FUNCTION_BLOCK CmdWaterDischargeSLBLogicBasic (* Basic Function Block Type *)
  (* Standard: 61499-2 *)
  (* Version 0.0, 7/31/2024, Administrator, Schneider Electric, Template *)
  PACKAGE SE.Nereda;
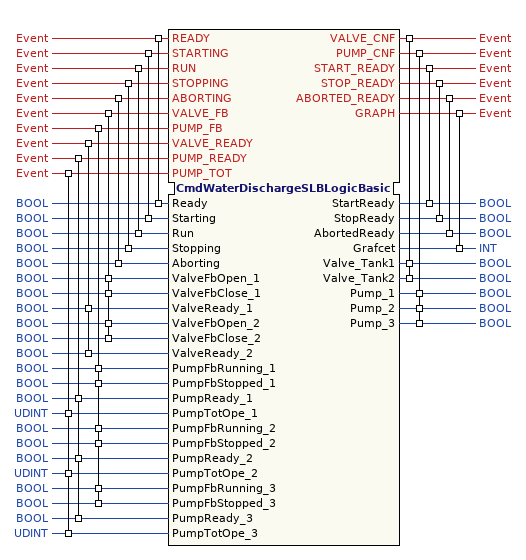
  EVENT_INPUT
    READY WITH Ready;
    STARTING WITH Starting; (* Normal Execution Request *)
    RUN WITH Run;
    STOPPING WITH Stopping;
    ABORTING WITH Aborting;
    VALVE_FB WITH ValveFbOpen_1, ValveFbClose_1, ValveFbOpen_2, ValveFbClose_2;
    PUMP_FB WITH PumpFbRunning_1, PumpFbStopped_1, PumpFbRunning_2, PumpFbStopped_2, PumpFbRunning_3, PumpFbStopped_3;
    VALVE_READY WITH ValveReady_1, ValveReady_2;
    PUMP_READY WITH PumpReady_1, PumpReady_2, PumpReady_3;
    PUMP_TOT WITH PumpTotOpe_1, PumpTotOpe_2, PumpTotOpe_3;
  END_EVENT
  EVENT_OUTPUT
    VALVE_CNF WITH Valve_Tank1, Valve_Tank2; (* Execution Confirmation *)
    PUMP_CNF WITH Pump_1, Pump_2, Pump_3;
    START_READY WITH StartReady;
    STOP_READY WITH StopReady;
    ABORTED_READY WITH AbortedReady;
    GRAPH WITH Grafcet;
  END_EVENT
  VAR_INPUT
    Ready : BOOL;
    Starting : BOOL; (* Input event qualifier *)
    Run : BOOL;
    Stopping : BOOL;
    Aborting : BOOL;
    ValveFbOpen_1 : BOOL;
    ValveFbClose_1 : BOOL;
    ValveReady_1 : BOOL;
    ValveFbOpen_2 : BOOL;
    ValveFbClose_2 : BOOL;
    ValveReady_2 : BOOL;
    PumpFbRunning_1 : BOOL;
    PumpFbStopped_1 : BOOL;
    PumpReady_1 : BOOL;
    PumpTotOpe_1 : UDINT;
    PumpFbRunning_2 : BOOL;
    PumpFbStopped_2 : BOOL;
    PumpReady_2 : BOOL;
    PumpTotOpe_2 : UDINT;
    PumpFbRunning_3 : BOOL;
    PumpFbStopped_3 : BOOL;
    PumpReady_3 : BOOL;
    PumpTotOpe_3 : UDINT;
  END_VAR
  VAR_OUTPUT
    StartReady : BOOL;
    StopReady : BOOL;
    AbortedReady : BOOL;
    Grafcet : INT;
    Valve_Tank1 : BOOL; (* Output event qualifier *)
    Valve_Tank2 : BOOL; (* Output event qualifier *)
    Pump_1 : BOOL;
    Pump_2 : BOOL;
    Pump_3 : BOOL;
  END_VAR
  VAR
    FirstPump : INT;
    SecondPump : INT;
  END_VAR
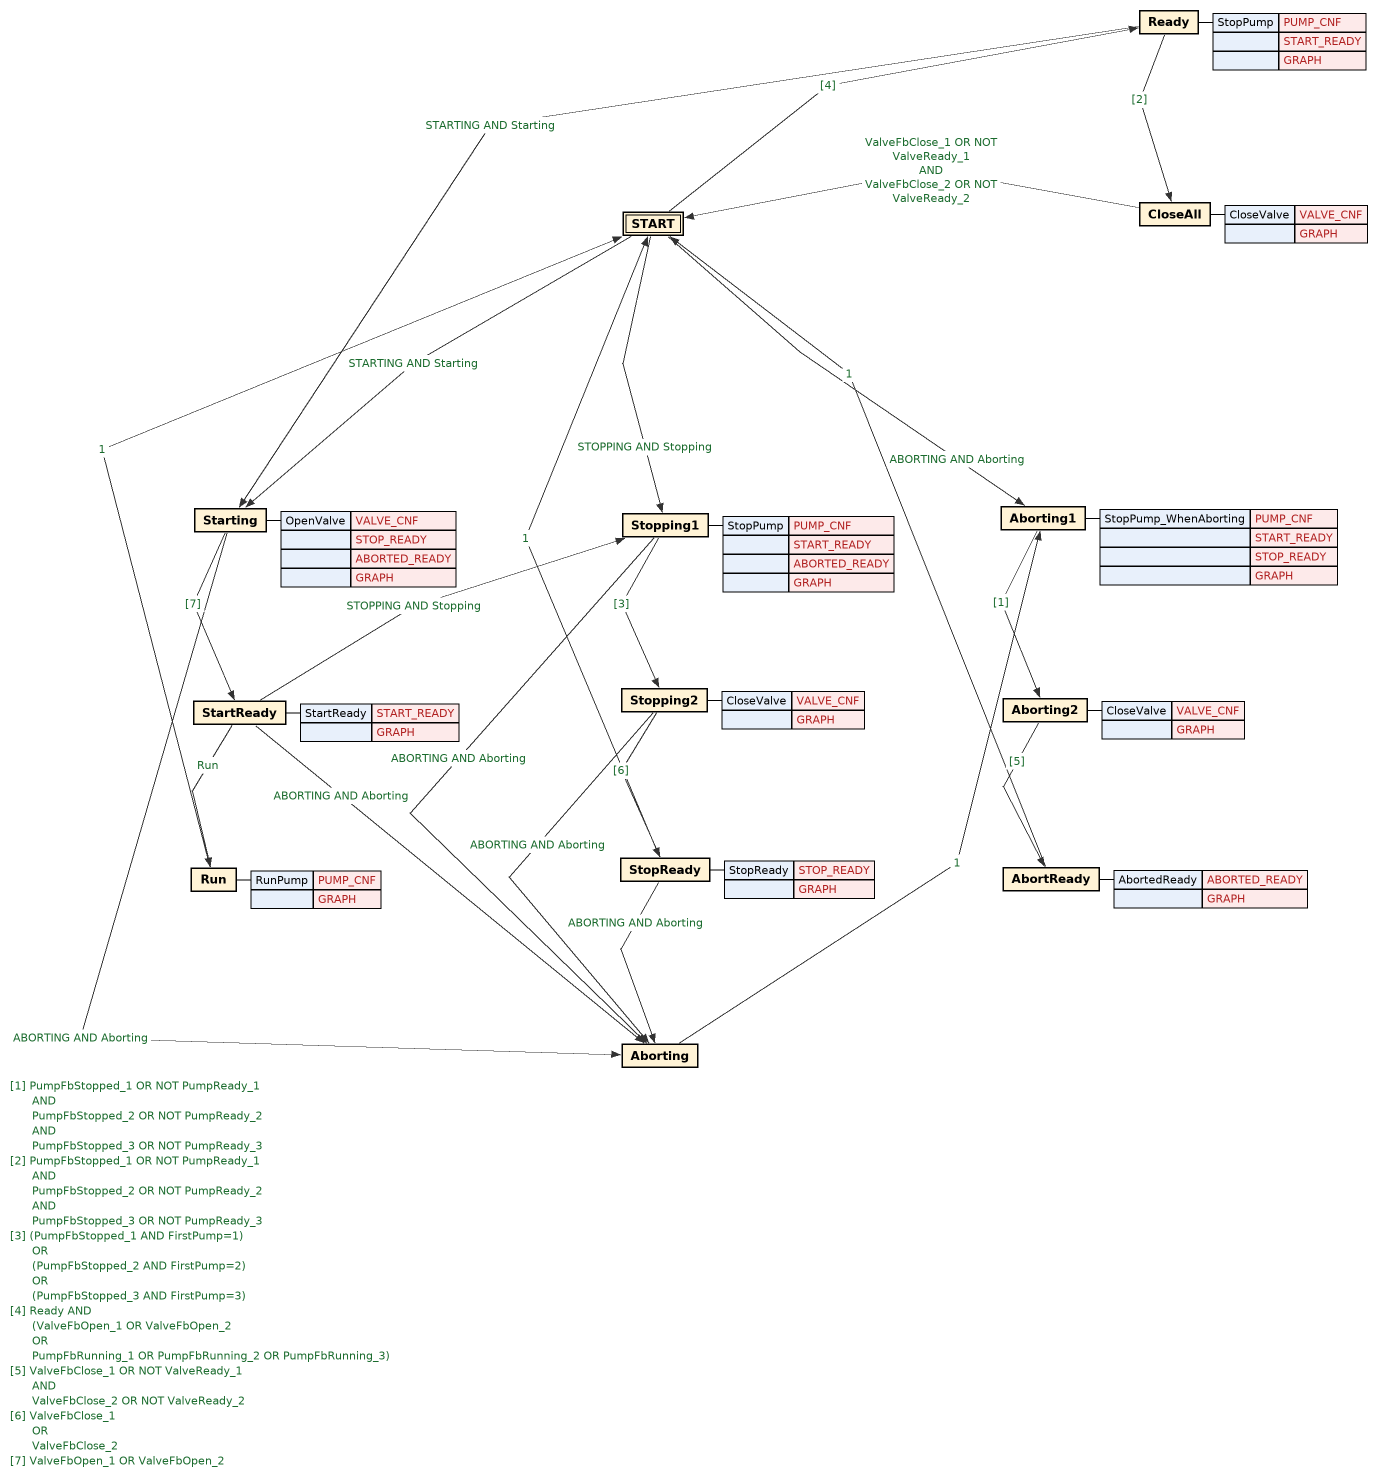
  EC_STATES
    START; (* Initial State *)
    Starting : OpenValve -> VALVE_CNF, -> STOP_READY, -> ABORTED_READY, -> GRAPH; (* Normal execution *)
    StartReady : StartReady -> START_READY, -> GRAPH;
    Stopping2 : CloseValve -> VALVE_CNF, -> GRAPH;
    StopReady : StopReady -> STOP_READY, -> GRAPH;
    Aborting2 : CloseValve -> VALVE_CNF, -> GRAPH;
    AbortReady : AbortedReady -> ABORTED_READY, -> GRAPH;
    Aborting;
    Ready : StopPump -> PUMP_CNF, -> START_READY, -> GRAPH;
    Run : RunPump -> PUMP_CNF, -> GRAPH;
    Aborting1 : StopPump_WhenAborting -> PUMP_CNF, -> START_READY, -> STOP_READY, -> GRAPH;
    Stopping1 : StopPump -> PUMP_CNF, -> START_READY, -> ABORTED_READY, -> GRAPH;
    CloseAll : CloseValve -> VALVE_CNF, -> GRAPH;
  END_STATES
  EC_TRANSITIONS
    START TO Starting := STARTING AND Starting;
    Starting TO StartReady := ValveFbOpen_1 OR ValveFbOpen_2;
    Run TO START := 1;
    START TO Stopping1 := STOPPING AND Stopping;
    Stopping2 TO StopReady := ValveFbClose_1 OR ValveFbClose_2;
    StopReady TO START := 1;
    Aborting2 TO AbortReady := ValveFbClose_1 OR NOT ValveReady_1 AND ValveFbClose_2 OR NOT ValveReady_2;
    START TO Aborting1 := ABORTING AND Aborting;
    AbortReady TO START := 1;
    Starting TO Aborting := ABORTING AND Aborting;
    Aborting TO Aborting1 := 1;
    Stopping2 TO Aborting := ABORTING AND Aborting;
    StopReady TO Aborting := ABORTING AND Aborting;
    START TO Ready := Ready AND (ValveFbOpen_1 OR ValveFbOpen_2 OR PumpFbRunning_1 OR PumpFbRunning_2 OR PumpFbRunning_3);
    CloseAll TO START := ValveFbClose_1 OR NOT ValveReady_1 AND ValveFbClose_2 OR NOT ValveReady_2;
    StartReady TO Run := Run;
    StartReady TO Aborting := ABORTING AND Aborting;
    Aborting1 TO Aborting2 := PumpFbStopped_1 OR NOT PumpReady_1 AND PumpFbStopped_2 OR NOT PumpReady_2 AND PumpFbStopped_3 OR NOT PumpReady_3;
    Stopping1 TO Stopping2 := (PumpFbStopped_1 AND FirstPump=1) OR (PumpFbStopped_2 AND FirstPump=2) OR (PumpFbStopped_3 AND FirstPump=3);
    Ready TO CloseAll := PumpFbStopped_1 OR NOT PumpReady_1 AND PumpFbStopped_2 OR NOT PumpReady_2 AND PumpFbStopped_3 OR NOT PumpReady_3;
    Stopping1 TO Aborting := ABORTING AND Aborting;
    Ready TO Starting := STARTING AND Starting;
    StartReady TO Stopping1 := STOPPING AND Stopping;
  END_TRANSITIONS
  ALGORITHM OpenValve IN ST: (* Normally executed algorithm *)
;
Grafcet := 1;
Valve_Tank1 := TRUE;
Valve_Tank2 := TRUE;
StopReady := FALSE;
AbortedReady := FALSE;
  END_ALGORITHM
  ALGORITHM StartReady IN ST:
;
Grafcet := 2;
StartReady := TRUE;
  END_ALGORITHM
  ALGORITHM CloseValve IN ST:
;
IF Grafcet = 4 THEN
	Grafcet := 5;
ELSIF Grafcet = 7 THEN
	Grafcet := 8;
END_IF;
Valve_Tank1 := FALSE;
Valve_Tank2 := FALSE;
  END_ALGORITHM
  ALGORITHM StopReady IN ST:
;
Grafcet := 6;
StopReady := TRUE;
  END_ALGORITHM
  ALGORITHM AbortedReady IN ST:
;
Grafcet := 9;
AbortedReady := TRUE;
  END_ALGORITHM
  ALGORITHM RunPump IN ST:
  VAR_TEMP
    FirstTOT : UDINT;
    SecondTOT : UDINT;
  END_VAR
;
Grafcet := 3;

(* Inicialização *)
FirstPump := 0;
SecondPump := 0;

FirstTOT := 16#FFFFFFFF;
SecondTOT := 16#FFFFFFFF;


(* Analisa Pump 1 *)
IF PumpReady_1 AND NOT PumpFbRunning_1 THEN

    IF PumpTotOpe_1 < FirstTOT THEN
        SecondTOT := FirstTOT;
        SecondPump := FirstPump;

        FirstTOT := PumpTotOpe_1;
        FirstPump := 1;

    ELSIF PumpTotOpe_1 < SecondTOT THEN
        SecondTOT := PumpTotOpe_1;
        SecondPump := 1;
    END_IF;

END_IF;


(* Analisa Pump 2 *)
IF PumpReady_2 AND NOT PumpFbRunning_2 THEN

    IF PumpTotOpe_2 < FirstTOT THEN
        SecondTOT := FirstTOT;
        SecondPump := FirstPump;

        FirstTOT := PumpTotOpe_2;
        FirstPump := 2;

    ELSIF PumpTotOpe_2 < SecondTOT THEN
        SecondTOT := PumpTotOpe_2;
        SecondPump := 2;
    END_IF;

END_IF;


(* Analisa Pump 3 *)
IF PumpReady_3 AND NOT PumpFbRunning_3 THEN

    IF PumpTotOpe_3 < FirstTOT THEN
        SecondTOT := FirstTOT;
        SecondPump := FirstPump;

        FirstTOT := PumpTotOpe_3;
        FirstPump := 3;

    ELSIF PumpTotOpe_3 < SecondTOT THEN
        SecondTOT := PumpTotOpe_3;
        SecondPump := 3;
    END_IF;

END_IF;


(* Limpa comandos *)
Pump_1 := FALSE;
Pump_2 := FALSE;
Pump_3 := FALSE;


(* Comanda as duas bombas selecionadas *)
IF StartReady THEN

    CASE FirstPump OF
        1: Pump_1 := TRUE;
        2: Pump_2 := TRUE;
        3: Pump_3 := TRUE;
    END_CASE;

    CASE SecondPump OF
        1: Pump_1 := TRUE;
        2: Pump_2 := TRUE;
        3: Pump_3 := TRUE;
    END_CASE;

END_IF;
  END_ALGORITHM
  ALGORITHM StopPump IN ST:
;
Grafcet := 4;
CASE FirstPump OF
	1: Pump_1 := FALSE;
	2: Pump_2 := FALSE;
	3: Pump_3 := FALSE;
END_CASE;

CASE SecondPump OF
	1: Pump_1 := FALSE;
	2: Pump_2 := FALSE;
	3: Pump_3 := FALSE;
END_CASE;


StartReady := FALSE;
AbortedReady  := FALSE;
  END_ALGORITHM
  ALGORITHM StopPump_WhenAborting IN ST:
;
Grafcet := 7;
Pump_1 := FALSE;
Pump_2 := FALSE;
Pump_3 := FALSE;
StartReady := FALSE;
StopReady := FALSE;
  END_ALGORITHM
END_FUNCTION_BLOCK
